// TIA Portal V16 export
// export: Created 2021-02-18T15:18:28.7030825Z, ExportSetting WithDefaults, DisplayName Totally Integrated Automation Portal, DisplayVersion V16 Update 3, DisplayName TIA Portal Version Control Interface, DisplayVersion V16 Update 2, DisplayName TIA Portal Openness, DisplayVersion V16 Update 3, DisplayName STEP 7 Professional, DisplayVersion V16 Update 3, DisplayName STEP 7 Safety, DisplayVersion V16, DisplayName WinCC Professional, DisplayVersion V16 Update 3
VAR_GLOBAL   // PLC tag table "PAL_SystemTags"
   _SysSignals01 AT %MB0 : Byte;   // System signals byte 01 — Logic and scan synchronised pulses   {ExternalWritable false}
   _False AT %M0.0 : Bool;   // System Logic Bit — Always FALSE   {ExternalWritable false}
   _True AT %M0.1 : Bool;   // System Logic Bit — Always TRUE   {ExternalWritable false}
   _50ms AT %M0.2 : Bool;   // System Timing — 50 ms pulse scan synchronised   {ExternalWritable false}
   _100ms AT %M0.3 : Bool;   // System Timing — 100 ms pulse scan synchronised   {ExternalWritable false}
   _200ms AT %M0.4 : Bool;   // System Timing — 200 ms pulse scan synchronised   {ExternalWritable false}
   _500ms AT %M0.5 : Bool;   // System Timing — 500 ms pulse scan synchronised   {ExternalWritable false}
   _1s AT %M0.6 : Bool;   // System Timing — 1 s pulse scan synchronised   {ExternalWritable false}
   _2s AT %M0.7 : Bool;   // System Timing — 2 s pulse scan synchronised   {ExternalWritable false}
   _SysSignals02 AT %MB1 : Byte;   // System signals byte 02 — scan signals and common square waves   {ExternalWritable false}
   _CycleTick AT %M1.0 : Bool;   // System Timing — Cycle tick (active odd cycles, alternates with _CycleTock)   {ExternalWritable false}
   _CycleTock AT %M1.1 : Bool;   // System Timing — Cycle tock (active even cycles, alternates with _CycleTick)   {ExternalWritable false}
   _CycleFirst AT %M1.2 : Bool;   // System Timing — First cycle detected   {ExternalWritable false}
   _100msSqW AT %M1.3 : Bool;   // System Timing — 100 ms square wave scan synchronised   {ExternalWritable false}
   _200msSqW AT %M1.4 : Bool;   // System Timing — 200 ms square wave scan synchronised   {ExternalWritable false}
   _500msSqW AT %M1.5 : Bool;   // System Timing — 500 ms square wave scan synchronised   {ExternalWritable false}
   _1sSqW AT %M1.6 : Bool;   // System Timing — 1 s square wave scan synchronised   {ExternalWritable false}
   _2sSqW AT %M1.7 : Bool;   // System Timing — 2 s square wave scan synchronised   {ExternalWritable false}
   _ClockMem AT %MB10 : Byte;   // Clock Memory (populated by the CPU)   {ExternalWritable false}
   _ClockMem_100msSqW AT %M10.0 : Bool;   // Clock Memory — 10.0 Hz square wave 0.1 s period   {ExternalWritable false}
   _ClockMem_200msSqW AT %M10.1 : Bool;   // Clock Memory — 5.00 Hz square wave 0.2 s period   {ExternalWritable false}
   _ClockMem_400msSqW AT %M10.2 : Bool;   // Clock Memory — 2.50 Hz square wave 0.4 s period   {ExternalWritable false}
   _ClockMem_500msSqW AT %M10.3 : Bool;   // Clock Memory — 2.00 Hz square wave 0.5 s period   {ExternalWritable false}
   _ClockMem_800msSqW AT %M10.4 : Bool;   // Clock Memory — 1.25 Hz square wave 0.8 s period   {ExternalWritable false}
   _ClockMem_1000msSqW AT %M10.5 : Bool;   // Clock Memory — 1.00 Hz square wave 1.0 s period   {ExternalWritable false}
   _ClockMem_1600msSqW AT %M10.6 : Bool;   // Clock Memory — 0.62 Hz square wave 1.6 s period   {ExternalWritable false}
   _ClockMem_2000msSqW AT %M10.7 : Bool;   // Clock Memory — 0.50 Hz square wave 2.0 s period   {ExternalWritable false}
   _SysSignals AT %MW0 : Int;   // System signals   {ExternalWritable false}
END_VAR
